FUNCTION_BLOCK GritScreenLogic (* CAT Function Block Type *)
  (* Standard: 61499-2 *)
  (* Version 0.0, 6/15/2026, Schneider Electric, template *)
  PACKAGE SE.Nereda;
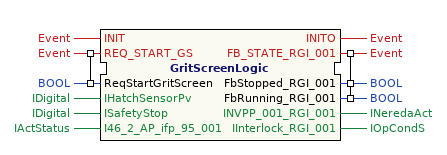
  EVENT_INPUT
    INIT;
    REQ_START_GS WITH ReqStartGritScreen;
  END_EVENT
  EVENT_OUTPUT
    INITO;
    FB_STATE_RGI_001 WITH FbStopped_RGI_001, FbRunning_RGI_001;
  END_EVENT
  VAR_INPUT
    ReqStartGritScreen : BOOL;
  END_VAR
  VAR_OUTPUT
    FbStopped_RGI_001 : BOOL;
    FbRunning_RGI_001 : BOOL;
  END_VAR
  SOCKETS
    IHatchSensorPv : IDigital;
    ISafetyStop : IDigital;
    I46_2_AP_ifp_95_001 : IActStatus;
  END_SOCKETS
  PLUGS
    INVPP_001_RGI_001 : INeredaAct;
  END_PLUGS
  PLUGS
    IInterlock_RGI_001 : IOpCondS; (* Condition summary chain output to downstream block *)
  END_PLUGS
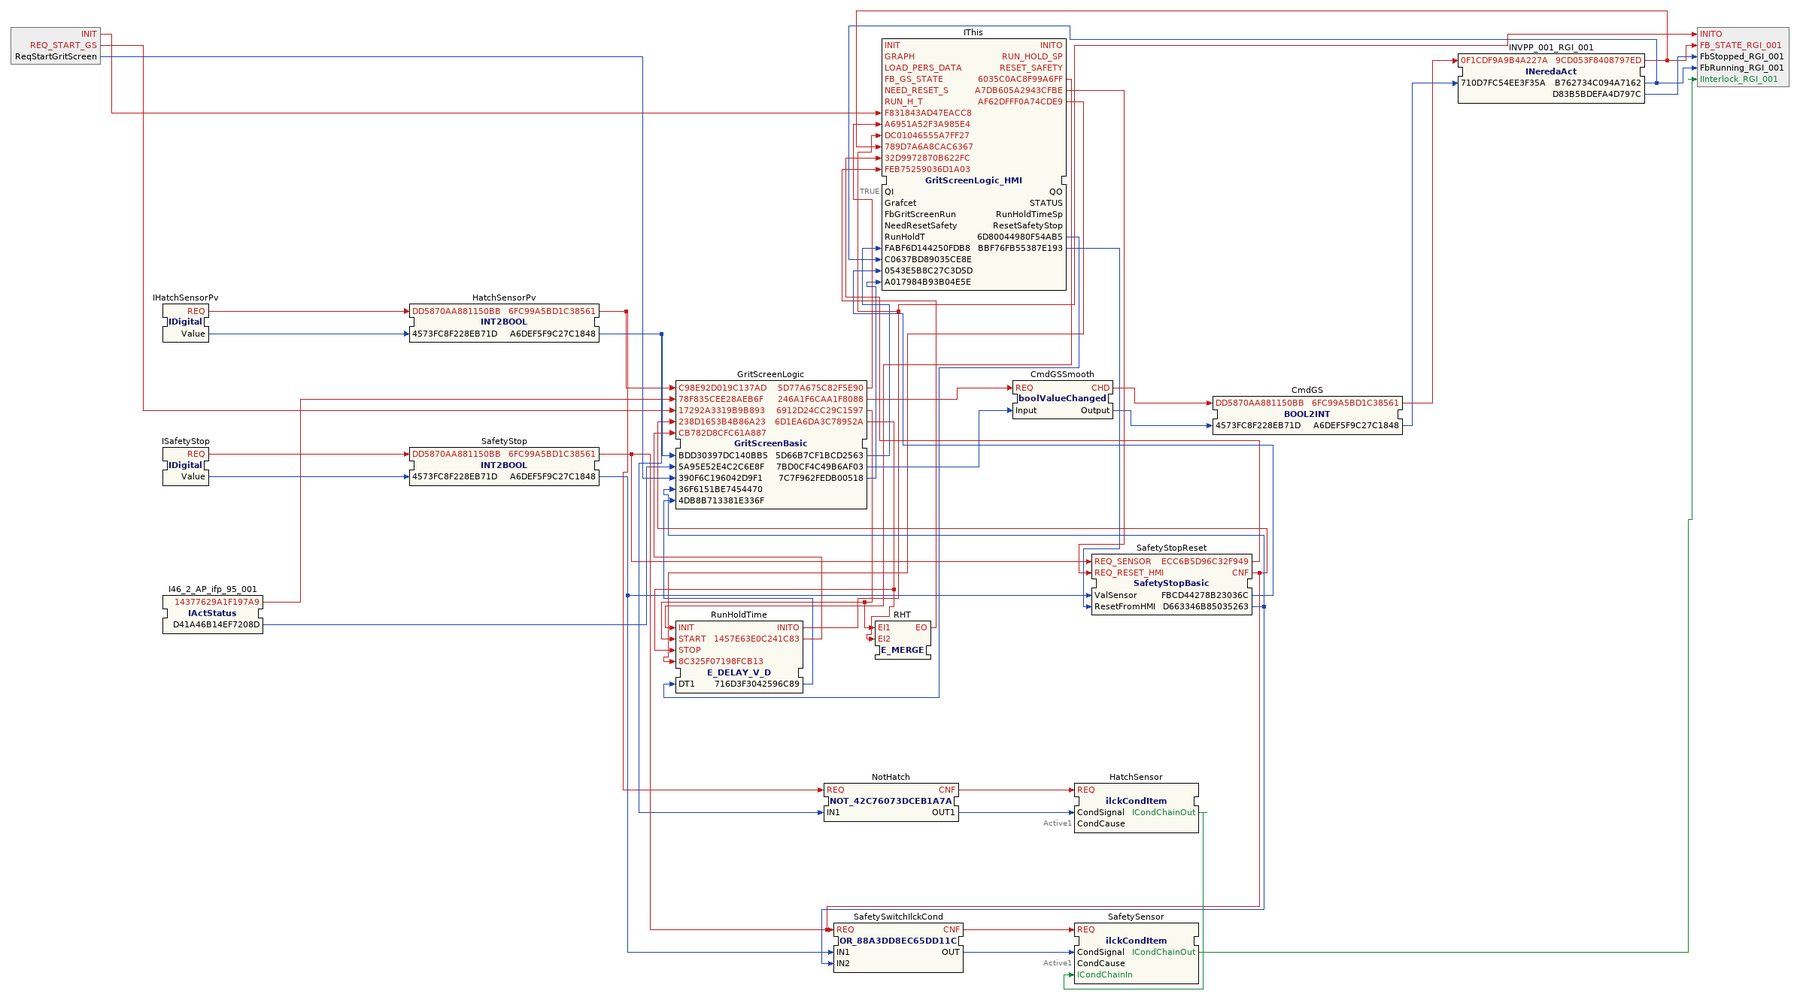
  (* 01 - FUNCTIONNAL INPUT INTERFACE *)
  (* 00 - INITIALIZATION *)
  (* 05 - LOGIC *)
  (* 03 - FIELD INTERFACE *)
  (* Grit Screen Logic *)
  (* 02 - FUNCTIONNAL OUTPUT INTERFACE *)
  (* 06 - HMI INTERFACE *)
  (* Interlock *)
  FBS
    GritScreenLogic : GritScreenBasic;
    RunHoldTime : E_DELAY_V_D;
    IThis : GritScreenLogic_HMI(QI := TRUE);
    CmdGSSmooth : boolValueChanged;
    SafetyStopReset : SafetyStopBasic;
    CmdGS : BOOL2INT;
    HatchSensorPv : INT2BOOL;
    SafetyStop : INT2BOOL;
    RHT : E_MERGE;
    HatchSensor : ilckCondItem(CondCause := Active1);
    SafetySensor : ilckCondItem(CondCause := Active1);
    NotHatch : NOT_42C76073DCEB1A7A; {SET_ATTRIBUTE(Configuration.GenericFBType.InterfaceParams, Runtime.Standard#CNT:=1;OUT${CNT$}:BOOL)}
    SafetySwitchIlckCond : OR_88A3DD8EC65DD11C; {SET_ATTRIBUTE(Configuration.GenericFBType.InterfaceParams, Runtime.Standard#CNT:=2;OUT:BOOL)}
  END_FBS
  EVENT_CONNECTIONS
    INIT TO IThis.F831843AD47EACC8;
    IHatchSensorPv.REQ TO HatchSensorPv.DD5870AA881150BB;
    ISafetyStop.REQ TO SafetyStop.DD5870AA881150BB;
    HatchSensorPv.6FC99A5BD1C38561 TO GritScreenLogic.C98E92D019C137AD;
    SafetyStop.6FC99A5BD1C38561 TO SafetyStopReset.REQ_SENSOR;
    I46_2_AP_ifp_95_001.14377629A1F197A9 TO GritScreenLogic.78F835CEE28AEB6F;
    REQ_START_GS TO GritScreenLogic.17292A3319B9B893;
    GritScreenLogic.5D77A675C82F5E90 TO IThis.A6951A52F3A985E4;
    RunHoldTime.INITO TO IThis.DC01046555A7FF27;
    INVPP_001_RGI_001.9CD053F8408797ED TO IThis.789D7A6A8CAC6367;
    SafetyStopReset.ECC6B5D96C32F949 TO IThis.32D9972870B622FC;
    IThis.6035C0AC8F99A6FF TO RunHoldTime.INIT;
    IThis.A7DB605A2943CFBE TO SafetyStopReset.REQ_RESET_HMI;
    SafetyStopReset.CNF TO GritScreenLogic.238D1653B4B86A23;
    RunHoldTime.1457E63E0C241C83 TO GritScreenLogic.CB782D8CFC61A887;
    GritScreenLogic.246A1F6CAA1F8088 TO CmdGSSmooth.REQ;
    GritScreenLogic.6912D24CC29C1597 TO RunHoldTime.START;
    GritScreenLogic.6D1EA6DA3C78952A TO RunHoldTime.STOP;
    CmdGSSmooth.CHD TO CmdGS.DD5870AA881150BB;
    CmdGS.6FC99A5BD1C38561 TO INVPP_001_RGI_001.0F1CDF9A9B4A227A;
    INVPP_001_RGI_001.9CD053F8408797ED TO FB_STATE_RGI_001;
    RunHoldTime.INITO TO INITO;
    IThis.AF62DFFF0A74CDE9 TO RunHoldTime.8C325F07198FCB13;
    GritScreenLogic.6912D24CC29C1597 TO RHT.EI1;
    GritScreenLogic.6D1EA6DA3C78952A TO RHT.EI2;
    RHT.EO TO IThis.FEB75259036D1A03;
    NotHatch.CNF TO HatchSensor.REQ;
    HatchSensorPv.6FC99A5BD1C38561 TO NotHatch.REQ;
    SafetyStop.6FC99A5BD1C38561 TO SafetySwitchIlckCond.REQ;
    SafetySwitchIlckCond.CNF TO SafetySensor.REQ;
    SafetyStopReset.CNF TO SafetySwitchIlckCond.REQ;
  END_CONNECTIONS
  DATA_CONNECTIONS
    IHatchSensorPv.Value TO HatchSensorPv.4573FC8F228EB71D;
    ISafetyStop.Value TO SafetyStop.4573FC8F228EB71D;
    HatchSensorPv.A6DEF5F9C27C1848 TO GritScreenLogic.BDD30397DC140BB5;
    SafetyStop.A6DEF5F9C27C1848 TO SafetyStopReset.ValSensor;
    I46_2_AP_ifp_95_001.D41A46B14EF7208D TO GritScreenLogic.5A95E52E4C2C6E8F;
    ReqStartGritScreen TO GritScreenLogic.390F6C196042D9F1;
    GritScreenLogic.5D66B7CF1BCD2563 TO IThis.FABF6D144250FDB8;
    INVPP_001_RGI_001.B762734C094A7162 TO IThis.C0637BD89035CE8E;
    SafetyStopReset.FBCD44278B23036C TO IThis.0543E5B8C27C3D5D;
    IThis.6D80044980F54AB5 TO RunHoldTime.DT1;
    IThis.BBF76FB55387E193 TO SafetyStopReset.ResetFromHMI;
    SafetyStopReset.D663346B85035263 TO GritScreenLogic.36F6151BE7454470;
    RunHoldTime.716D3F3042596C89 TO GritScreenLogic.4DB8B713381E336F;
    GritScreenLogic.7BD0CF4C49B6AF03 TO CmdGSSmooth.Input;
    CmdGSSmooth.Output TO CmdGS.4573FC8F228EB71D;
    CmdGS.A6DEF5F9C27C1848 TO INVPP_001_RGI_001.710D7FC54EE3F35A;
    INVPP_001_RGI_001.D83B5BDEFA4D797C TO FbStopped_RGI_001;
    INVPP_001_RGI_001.B762734C094A7162 TO FbRunning_RGI_001;
    GritScreenLogic.7C7F962FEDB00518 TO IThis.A017984B93B04E5E;
    NotHatch.OUT1 TO HatchSensor.CondSignal;
    HatchSensorPv.A6DEF5F9C27C1848 TO NotHatch.IN1;
    SafetyStop.A6DEF5F9C27C1848 TO SafetySwitchIlckCond.IN1;
    SafetySwitchIlckCond.OUT TO SafetySensor.CondSignal;
    SafetyStopReset.D663346B85035263 TO SafetySwitchIlckCond.IN2;
  END_CONNECTIONS
  ADAPTER_CONNECTIONS
    HatchSensor.ICondChainOut TO SafetySensor.ICondChainIn;
    SafetySensor.ICondChainOut TO IInterlock_RGI_001;
  END_CONNECTIONS
END_FUNCTION_BLOCK
